# B&R Automation Studio project ProyectoDardos
Automation Studio 4.9

## Configuration Config1

CPU 4PPC70.0702-23B, AutomationRuntime B4.92, Build 4.1.2, Vc V4.72.5

### Task classes (Cpu.sw)
```
Cyclic#4:
  VisuCtrl <- Visu.VisuCtrl.prg
  ScoreCtrl <- Source.ScoreCtrl.prg
Cyclic#5 (cycle 250000 us, tolerance 250000 us):
  VisapiCtrl <- Source.VisapiCtrl.prg
VcDataObjects: VisuDa <- Visu.VisuDardos.dob
Binaries: vcnet, vccdbox, udbdef, vcrt, vcpkat, vcctext, vccurl, vcchtml, vccslider, visvc, vcfile, vcgclass, vccstr, vcpdsw, vccshape, arial, vccbmp, vcmgr, vcdsloc, VisuDa01, vcfntttf, vccovl, vcshared, arialbd, VisuDa02, VisuDa03, vcalarm, vccdt, vccline, vcpfar00, vccbtn, vcpdvnc, vcbclass, vcxml, vcdsint, vctcal, TCData, FWRules, vccnum, sysconf, iomap, asfw, Role, ashwac, ashwd, User, arconfig
Libraries: visapi, standard, vcresman, asieccon, fileio, astime, runtime, dataobj
```

### Hardware
```
4PPC70_0702_23B : 4PPC70.0702-23B v1.5.4.0
  Connector IF2:
    ActivateDevice = 1
    Mode = Manual
    InternetAddress = 192.168.150.95
    SubnetMask = 255.255.255.0
    Vnc1
    VncVcObjectName1 = VisuDa
    VncKeyMappingFile1 = VC\PS2-Keyboard.dis
    ActivateSnmp = 2
  ConfigurationID = proyectoDardos_Config1
  Cyclic5Duration = 250000
  Cyclic5Tolerance = 250000
  FileDevice1
  FileDeviceName1 = USER
  FileDevicePath1 = USER_PATH
  VcObjectName = VisuDa
  KeyMappingFile = VC\4PPC70_0702_23B.dis
```

## Logical view

### Global.typ - Global data types
```iecst
(*gMainCtrl_type*)

TYPE
	gMainCtrl_type : 	STRUCT
		visapiCtrl : visapiCtrl_type;
		scoreCtrl : scoreCtrl_type;
	END_STRUCT;
END_TYPE

(*visapiCtrl_type*)

TYPE
	visapiCtrl_type : 	STRUCT
		cmd : visapiCtrl_cmd_type;
		status : visapiCtrl_status_type;
		state : visapiCtrl_state_type;
	END_STRUCT;
	visapiCtrl_cmd_type : 	STRUCT
		readyToDraw : BOOL;
	END_STRUCT;
	visapiCtrl_status_type : 	STRUCT
		touchCoordinateX : REAL;
		drawing : BOOL;
		touchCoordinateY : REAL;
		valitTouch : BOOL;
		homeYCoordenate : REAL;
		homeXCoordenate : REAL;
		widthEllipse : ARRAY[1..6]OF UINT;
		heigthEllipse : ARRAY[1..6]OF UINT;
		widthTarget : UDINT;
		heigthTarget : UDINT;
		touchCoordinateStatus : BOOL;
		widthRect : UDINT;
	END_STRUCT;
	visapiCtrl_state_type :
		(
		WAIT := 0,
		DRAWING := 10,
		ERROR := 100
		);
END_TYPE

(*scoreCtrl_type*)

TYPE
	scoreCtrl_type : 	STRUCT
		cmd : scoreCtrl_cmd_type;
		status : scoreCtrl_status_type;
		state : scoreCtrl_state_type;
	END_STRUCT;
	scoreCtrl_cmd_type : 	STRUCT
		addPointScore : BOOL;
	END_STRUCT;
	scoreCtrl_status_type : 	STRUCT
		validTouch : BOOL;
		additivePoint : ARRAY[1..MAX_RADIUS_WITH_TARGET]OF UINT;
		incorrectScore : BOOL;
		correctScore : BOOL;
		cumulateScore : UINT;
		cumulateShots : UINT;
	END_STRUCT;
	scoreCtrl_state_type :
		(
		WAIT_SCORE := 0,
		GET_SCORE := 10,
		ERROR_SCORE := 100
		);
END_TYPE

(*gMachinePar*)

TYPE
	gMachinePar_type : 	STRUCT
		New_Member : USINT;
	END_STRUCT;
END_TYPE

(*gVisuCtrl_type*)

TYPE
	gVisuCtrl_type : 	STRUCT
		numInput : gVIsu_numInput_type;
		runtime : gVisu_runtime_type;
		button : gVisu_button_type;
		textOutput : gVisu_textOutput_type;
	END_STRUCT;
	gVIsu_numInput_type : 	STRUCT
		radiusWidth : ARRAY[1..MAX_RADIUS_WITH_TARGET]OF UINT;
		selectedRadiusWidth : ARRAY[1..MAX_RADIUS_WITH_TARGET]OF UINT;
	END_STRUCT;
	gVisu_runtime_type : 	STRUCT
		showButtonStartNewGame : USINT;
	END_STRUCT;
	gVisu_button_type : 	STRUCT
		startNewGame : BOOL;
	END_STRUCT;
	gVisu_textOutput_type : 	STRUCT
		statusGame : USINT;
	END_STRUCT;
END_TYPE
```

### Global.var - Global variables
```iecst
VAR
	gMainCtrl : gMainCtrl_type;
END_VAR
VAR RETAIN
	gMachinePar : {REDUND_UNREPLICABLE} gMachinePar_type := (0);
END_VAR
VAR CONSTANT
	LEFT_OFFSET : UINT := 28;
	TOP_OFFSET : UINT := 60;
	MAX_X_COORDINATE : UDINT := 434;
	MAX_Y_COORDINATE : UDINT := 413;
	MIN_X_COORDINATE : UDINT := 28;
	MIN_Y_COORDINATE : UDINT := 60;
	MAX_RADIUS : INT := 6;
	MAX_RADIUS_WITH_TARGET : UINT := 7;
END_VAR
VAR
	gVisuCtrl : gVisuCtrl_type;
END_VAR
VAR CONSTANT
	COORDENATE_Y_BITMAP : INT := 62;
	COORDENATE_X_BITMAP : INT := 358;
	MAX_SCORE : INT := 500;
	MAX_SHOTS : INT := 10;
END_VAR
```

### Program Logical/Source/ScoreCtrl (IEC)

#### Variables.var
```iecst
VAR
	getTouch : BOOL;
	homeXCoordenate : REAL;
	pointValue : UINT;
	ratio : REAL;
	homeYCoordenate : REAL;
	firstProduct : REAL;
	secondProduct : REAL;
END_VAR
VAR CONSTANT
	EXPONENT : INT := 2;
END_VAR
VAR
	intRatio : INT;
	countPointValue : UINT;
	valitPoint : BOOL;
	newTouch : BOOL;
	addPointsReady : BOOL;
	remainingShots : USINT;
END_VAR
VAR RETAIN
	maxShots : USINT;
	maxCountPointValue : INT;
END_VAR
VAR
	validCoordenate : BOOL;
	restorePointValues : BOOL;
	confirmValueRadius : BOOL;
END_VAR
(*AJUSTE DE PUNTAJES*)
VAR
	i : INT;
	actualRadius : INT;
	nextRadius : BOOL;
	previusRadius : BOOL;
	addivePoint : UINT;
END_VAR
```

#### Main.st
```iecst
PROGRAM _INIT
	actualRadius := 1;
	gMainCtrl.scoreCtrl.status.additivePoint[1] := 100;
	gMainCtrl.scoreCtrl.status.additivePoint[2] := 80;
	gMainCtrl.scoreCtrl.status.additivePoint[3] := 60;
	gMainCtrl.scoreCtrl.status.additivePoint[4] := 40;
	gMainCtrl.scoreCtrl.status.additivePoint[5] := 20;
	gMainCtrl.scoreCtrl.status.additivePoint[6] := 10;
	gMainCtrl.scoreCtrl.status.additivePoint[7] := 5;

END_PROGRAM

PROGRAM _CYCLIC
	homeXCoordenate := (gMainCtrl.visapiCtrl.status.homeXCoordenate);
	homeYCoordenate	:= (gMainCtrl.visapiCtrl.status.homeYCoordenate);
	newTouch		:= 	gMainCtrl.visapiCtrl.status.touchCoordinateStatus;

	firstProduct 	:= ABS(homeXCoordenate - gMainCtrl.visapiCtrl.status.touchCoordinateX);
	secondProduct	:= ABS(homeYCoordenate - gMainCtrl.visapiCtrl.status.touchCoordinateY);
	ratio := SQRT(EXPT(firstProduct,EXPONENT)+(EXPT(secondProduct,EXPONENT)));
	intRatio := REAL_TO_INT(ratio);

	IF restorePointValues THEN
		gMainCtrl.scoreCtrl.status.additivePoint[1] := 10;
		gMainCtrl.scoreCtrl.status.additivePoint[2] := 20;
		gMainCtrl.scoreCtrl.status.additivePoint[3] := 30;
		gMainCtrl.scoreCtrl.status.additivePoint[4] := 10;
		gMainCtrl.scoreCtrl.status.additivePoint[5] := 10;
		gMainCtrl.scoreCtrl.status.additivePoint[6] := 10;
		gMainCtrl.scoreCtrl.status.additivePoint[7] := 10;
	END_IF;

	///// AJUSTES DE PUNTAJE PARA CADA CIRCUNFERENCIA
	IF (actualRadius >= 1) AND (actualRadius <7) THEN
		IF EDGEPOS(nextRadius) THEN
			actualRadius:= actualRadius + 1;
		END_IF;
	END_IF;
	IF (actualRadius > 1) AND (actualRadius <= 7) THEN
		IF EDGEPOS(previusRadius) THEN
			actualRadius:= actualRadius - 1;
		END_IF;
	END_IF;

	IF actualRadius = 1 AND confirmValueRadius THEN
		confirmValueRadius := FALSE;
		gMainCtrl.scoreCtrl.status.additivePoint[1] := addivePoint;
	ELSIF actualRadius = 2 AND confirmValueRadius THEN
		confirmValueRadius := FALSE;
		gMainCtrl.scoreCtrl.status.additivePoint[2] := addivePoint;
	ELSIF actualRadius = 3 AND confirmValueRadius THEN
		confirmValueRadius := FALSE;
		gMainCtrl.scoreCtrl.status.additivePoint[3] := addivePoint;
	ELSIF actualRadius = 4 AND confirmValueRadius THEN
		confirmValueRadius := FALSE;
		gMainCtrl.scoreCtrl.status.additivePoint[4] := addivePoint;
	ELSIF actualRadius = 5 AND confirmValueRadius THEN
		confirmValueRadius := FALSE;
		gMainCtrl.scoreCtrl.status.additivePoint[5] := addivePoint;
	ELSIF actualRadius = 6 AND confirmValueRadius THEN
		confirmValueRadius := FALSE;
		gMainCtrl.scoreCtrl.status.additivePoint[6] := addivePoint;
	ELSIF actualRadius = 7 AND confirmValueRadius THEN
		confirmValueRadius := FALSE;
		gMainCtrl.scoreCtrl.status.additivePoint[7] := addivePoint;
	END_IF;

	IF	gMainCtrl.visapiCtrl.status.valitTouch THEN
		validCoordenate := TRUE;
	ELSE
		validCoordenate := FALSE;
	END_IF;

	CASE gMainCtrl.scoreCtrl.state OF

		WAIT_SCORE:

			IF EDGEPOS(newTouch) THEN
				IF (intRatio < gMainCtrl.visapiCtrl.status.widthRect) THEN
					gMainCtrl.scoreCtrl.cmd.addPointScore := TRUE;
					gMainCtrl.scoreCtrl.state	 := GET_SCORE;
				END_IF;
			END_IF;

		GET_SCORE:

			IF gMainCtrl.scoreCtrl.status.cumulateShots <= (MAX_SHOTS-1) AND gMainCtrl.scoreCtrl.cmd.addPointScore AND (gMainCtrl.scoreCtrl.status.cumulateScore < MAX_SCORE) AND validCoordenate THEN
				IF (intRatio <= gMainCtrl.visapiCtrl.status.heigthEllipse[1]/2) AND (intRatio > gMainCtrl.visapiCtrl.status.heigthEllipse[2]/2)  THEN
					gMainCtrl.scoreCtrl.cmd.addPointScore := FALSE;
					gMainCtrl.scoreCtrl.status.cumulateScore := gMainCtrl.scoreCtrl.status.cumulateScore  + gMainCtrl.scoreCtrl.status.additivePoint[7];
				ELSIF (intRatio <= gMainCtrl.visapiCtrl.status.heigthEllipse[2]/2) AND (intRatio > gMainCtrl.visapiCtrl.status.heigthEllipse[3]/2)  THEN
					gMainCtrl.scoreCtrl.cmd.addPointScore := FALSE;
					gMainCtrl.scoreCtrl.status.cumulateScore := gMainCtrl.scoreCtrl.status.cumulateScore + gMainCtrl.scoreCtrl.status.additivePoint[6];
				ELSIF (intRatio <= gMainCtrl.visapiCtrl.status.heigthEllipse[3]/2) AND (intRatio > gMainCtrl.visapiCtrl.status.heigthEllipse[4]/2)  THEN
					gMainCtrl.scoreCtrl.cmd.addPointScore := FALSE;
					pointValue := gMainCtrl.scoreCtrl.status.additivePoint[5];
					gMainCtrl.scoreCtrl.status.cumulateScore := gMainCtrl.scoreCtrl.status.cumulateScore + pointValue;
				ELSIF (intRatio <= gMainCtrl.visapiCtrl.status.heigthEllipse[4]/2) AND (intRatio > gMainCtrl.visapiCtrl.status.heigthEllipse[5]/2)  THEN
					gMainCtrl.scoreCtrl.cmd.addPointScore := FALSE;
					pointValue := gMainCtrl.scoreCtrl.status.additivePoint[4];
					gMainCtrl.scoreCtrl.status.cumulateScore := gMainCtrl.scoreCtrl.status.cumulateScore + pointValue;
				ELSIF (intRatio <= gMainCtrl.visapiCtrl.status.heigthEllipse[5]/2) AND (intRatio > gMainCtrl.visapiCtrl.status.heigthEllipse[6]/2)  THEN
					gMainCtrl.scoreCtrl.cmd.addPointScore := FALSE;
					pointValue := gMainCtrl.scoreCtrl.status.additivePoint[3];
					gMainCtrl.scoreCtrl.status.cumulateScore := gMainCtrl.scoreCtrl.status.cumulateScore + pointValue;
				ELSIF (intRatio <= gMainCtrl.visapiCtrl.status.heigthEllipse[6]/2) AND (intRatio > gMainCtrl.visapiCtrl.status.heigthTarget/2)  THEN
					gMainCtrl.scoreCtrl.cmd.addPointScore := FALSE;
					pointValue := gMainCtrl.scoreCtrl.status.additivePoint[2];
					gMainCtrl.scoreCtrl.status.cumulateScore := gMainCtrl.scoreCtrl.status.cumulateScore + pointValue;
				ELSIF (intRatio <= gMainCtrl.visapiCtrl.status.heigthTarget/2)  THEN
					gMainCtrl.scoreCtrl.cmd.addPointScore := FALSE;
					pointValue := gMainCtrl.scoreCtrl.status.additivePoint[1];
					gMainCtrl.scoreCtrl.status.cumulateScore := gMainCtrl.scoreCtrl.status.cumulateScore + pointValue;
				ELSIF (intRatio > gMainCtrl.visapiCtrl.status.heigthEllipse[1]/2) AND (gMainCtrl.scoreCtrl.cmd.addPointScore )(* AND (gMainCtrl.scoreCtrl.status.cumulateShots <= (MAX_SHOTS-1))*) THEN
					gMainCtrl.scoreCtrl.cmd.addPointScore := FALSE;
				END_IF;

				gMainCtrl.scoreCtrl.status.cumulateShots := gMainCtrl.scoreCtrl.status.cumulateShots + 1;

			END_IF;

			IF 	intRatio > (gMainCtrl.visapiCtrl.status.heigthEllipse[1]/2) THEN
				gMainCtrl.scoreCtrl.status.incorrectScore := TRUE;
				gMainCtrl.scoreCtrl.status.correctScore := FALSE;
			ELSIF (intRatio <= gMainCtrl.visapiCtrl.status.heigthEllipse[1]/2) THEN
				gMainCtrl.scoreCtrl.status.correctScore := TRUE;
				gMainCtrl.scoreCtrl.status.incorrectScore := FALSE;
			END_IF

			IF EDGENEG(newTouch) THEN
				gMainCtrl.scoreCtrl.state	 := WAIT_SCORE;
			END_IF;

	END_CASE;

END_PROGRAM

PROGRAM _EXIT
			(* Insert code here *)

END_PROGRAM
```

### Program Logical/Source/VisapiCtrl (IEC)

#### Types.typ
```iecst
TYPE
	VA_SetupX_0 : 	STRUCT
		enable : BOOL;
		VCHandle : VCHANDLE;
		interpreter : STRING[80] := 'VisuDa';
		status : UINT;
	END_STRUCT;
	VA_Saccess_0 : 	STRUCT
		enable : BOOL;
		VCHandle : VCHANDLE;
		status : UINT;
	END_STRUCT;
END_TYPE
```

#### Variables.var
```iecst
(*VISAPI*)
VAR
	ready : UINT;
	VC_HANDLE : UDINT;
	interpreter : STRING[80] := 'VisuDa';
END_VAR
(*VA_Rect*)
VAR
	xRect : ARRAY[1..MAX_RECT] OF UINT := [28,0,229]; (*coordenada X del rectangulo*)
	yRect : ARRAY[1..MAX_RECT] OF UINT := [60,235,0]; (*coordenada Y del rectangulo*)
	widthRect : ARRAY[1..MAX_RECT] OF UINT := [406,0,4]; (*ancho del rectangulo*)
	heigthRect : ARRAY[1..MAX_RECT] OF UINT := [353,4,0]; (*altura del rectangulo*)
	fillRect : ARRAY[1..MAX_RECT] OF UINT := [255,2(45)]; (*relleno del rectangulo*)
	colorRect : ARRAY[1..MAX_RECT] OF UINT := [255,2(45)]; (*contorno del rectanculo*)
END_VAR
(*VA_Ellipse*)
VAR CONSTANT
	xEllipse : UINT := 231; (*coordenada X de la elipse*)
	yEllipse : UINT := 237; (*coordenadas Y de la elipse*)
END_VAR
VAR RETAIN
	heigthEllipse : ARRAY[1..MAX_RADIUS] OF UINT; (*altura de la elipse*)
	widthEllipse : ARRAY[1..MAX_RADIUS] OF UINT; (*ancho de la elipse*)
END_VAR
VAR
	fillEllipse : ARRAY[1..MAX_RADIUS] OF UINT := [45,16,45,16,45,16]; (*relleno de la elipse*)
END_VAR
VAR RETAIN
	colorEllipse : ARRAY[1..MAX_RADIUS] OF UINT := [0,16,45,16,45,16]; (*contorno de la elipse*)
END_VAR
VAR CONSTANT
	xTarget : UINT := 231; (*coordenada X del target*)
	yTarget : UINT := 237; (*coordenada Y del target*)
END_VAR
VAR
	heigthTarget : UINT;
	widthTarget : UINT;
	fillTarget : USINT := 205;
	colorTarget : USINT := 45;
	updateRadio : UINT;
END_VAR
(*AUX *)
VAR
	actualPage : UINT; (*pagina actual*)
	j : INT;
	defaultRadiusValues : BOOL;
END_VAR
VAR CONSTANT
	MAX_RECT : INT := 3;
END_VAR
(*VA_GetTouchAction*)
VAR
	xTouchPosition : UDINT;
	yTouchPosition : UDINT;
	Touch : TouchAction;
	newTouch : BOOL;
	changeRatioValue : BOOL;
	actualRadius : INT;
	nextRadius : BOOL;
	previusRadius : BOOL;
	confirmValueRadius : BOOL;
END_VAR
```

#### Main.st
```iecst
PROGRAM _INIT
	//Inicialización de circunferencias
	gMainCtrl.visapiCtrl.status.heigthEllipse[1] := 330;
	gMainCtrl.visapiCtrl.status.heigthEllipse[2] := 280;
	gMainCtrl.visapiCtrl.status.heigthEllipse[3] := 230;
	gMainCtrl.visapiCtrl.status.heigthEllipse[4] := 180;
	gMainCtrl.visapiCtrl.status.heigthEllipse[5] := 130;
	gMainCtrl.visapiCtrl.status.heigthEllipse[6] := 80;
	gMainCtrl.visapiCtrl.status.heigthTarget	 := 40;
	heigthTarget	 := 30;
	xTouchPosition;
	yTouchPosition;
	actualRadius := 1;
END_PROGRAM

PROGRAM _CYCLIC

	FOR j:= 1 TO MAX_RADIUS DO
		heigthEllipse[j] := gMainCtrl.visapiCtrl.status.heigthEllipse[j];
		widthEllipse[j] := gMainCtrl.visapiCtrl.status.widthEllipse[j];
	END_FOR;

	//CORDENADAS, ALTO Y ANCHO DE LOS RECTANGULOS QUE DIVIDEN EL TABLERO
	xRect[2]:= ((widthRect[1]/2)-(gMainCtrl.visapiCtrl.status.widthEllipse[1]/2))+ LEFT_OFFSET;
	yRect[3]:=((heigthRect[1]/2)-(gMainCtrl.visapiCtrl.status.widthEllipse[1]/2))+ TOP_OFFSET;
	widthRect[2] := gMainCtrl.visapiCtrl.status.widthEllipse[1];
	heigthRect[3] := gMainCtrl.visapiCtrl.status.widthEllipse[1];
	widthTarget	:= heigthTarget;

	IF defaultRadiusValues THEN
		gMainCtrl.visapiCtrl.status.heigthEllipse[1] := 330;
		gMainCtrl.visapiCtrl.status.heigthEllipse[2] := 280;
		gMainCtrl.visapiCtrl.status.heigthEllipse[3] := 230;
		gMainCtrl.visapiCtrl.status.heigthEllipse[4] := 180;
		gMainCtrl.visapiCtrl.status.heigthEllipse[5] := 130;
		gMainCtrl.visapiCtrl.status.heigthEllipse[6] := 80;
		gMainCtrl.visapiCtrl.status.heigthTarget	 := 40;
	END_IF;

	IF Touch.status = 1 THEN
		newTouch 	:= TRUE;
	ELSE
		newTouch	:= FALSE;
	END_IF;

	///// AJUSTES DE PUNTAJE PARA CADA CIRCUNFERENCIA
	IF (actualRadius >= 1) AND (actualRadius <7) THEN
		IF EDGEPOS(nextRadius) THEN
			actualRadius:= actualRadius + 1;
		END_IF;
	END_IF;
	IF (actualRadius > 1) AND (actualRadius <= 7) THEN
		IF EDGEPOS(previusRadius) THEN
			actualRadius:= actualRadius - 1;
		END_IF;
	END_IF;

	IF actualRadius = 1 AND confirmValueRadius THEN
		confirmValueRadius := FALSE;
		heigthTarget		:= updateRadio;
	ELSIF actualRadius = 2 AND confirmValueRadius THEN
		confirmValueRadius := FALSE;
		gMainCtrl.visapiCtrl.status.heigthEllipse[6] := updateRadio;
	ELSIF actualRadius = 3 AND confirmValueRadius THEN
		confirmValueRadius := FALSE;
		gMainCtrl.visapiCtrl.status.heigthEllipse[5] := updateRadio;
	ELSIF actualRadius = 4 AND confirmValueRadius THEN
		confirmValueRadius := FALSE;
		gMainCtrl.visapiCtrl.status.heigthEllipse[4] := updateRadio;
	ELSIF actualRadius = 5 AND confirmValueRadius THEN
		confirmValueRadius := FALSE;
		gMainCtrl.visapiCtrl.status.heigthEllipse[3] := updateRadio;
	ELSIF actualRadius = 6 AND confirmValueRadius THEN
		confirmValueRadius := FALSE;
		gMainCtrl.visapiCtrl.status.heigthEllipse[2] := updateRadio;
	ELSIF actualRadius = 7 AND confirmValueRadius THEN
		confirmValueRadius := FALSE;
		gMainCtrl.visapiCtrl.status.heigthEllipse[1] := updateRadio;
	END_IF;

	CASE gMainCtrl.visapiCtrl.state OF

		WAIT:
			IF ready <> 1 THEN
				VC_HANDLE := VA_Setup(1,interpreter);
				ready := 1;
			END_IF;
			IF  (*oldHeight <> height AND*) ready = 1 THEN
				gMainCtrl.visapiCtrl.state := DRAWING;
			END_IF;

		DRAWING:

			IF ready = 1 AND actualPage = 0 THEN
				IF VA_Saccess(1, VC_HANDLE) = 0 THEN

					IF changeRatioValue THEN
						changeRatioValue	:= FALSE;
						VA_Redraw(1,VC_HANDLE);
					END_IF;

					VA_Rect(1,VC_HANDLE,xRect[1],yRect[1],widthRect[1],heigthRect[1],fillRect[1],colorRect[1]);

					FOR j:= 1 TO (MAX_RADIUS) DO
						fillEllipse[j+1]	:= colorEllipse[j+1];
						gMainCtrl.visapiCtrl.status.widthEllipse[j] := gMainCtrl.visapiCtrl.status.heigthEllipse[j];
						VA_Ellipse(1,VC_HANDLE,xEllipse ,yEllipse,gMainCtrl.visapiCtrl.status.heigthEllipse[j] ,gMainCtrl.visapiCtrl.status.widthEllipse[j],fillEllipse[j],colorEllipse[j]);
					END_FOR;

					VA_Rect(1,VC_HANDLE,xRect[2],yRect[2],widthRect[2],heigthRect[2],fillRect[2],colorRect[2]); //RECTANGULO HORIZONTAL
					VA_Rect(1,VC_HANDLE,xRect[3],yRect[3],widthRect[3],heigthRect[3],fillRect[3],colorRect[3]); //RECTANGULO VERTICAL
					VA_Ellipse(1,VC_HANDLE,xTarget,yTarget,heigthTarget,widthTarget,fillTarget,colorTarget); //TARGET
					VA_GetTouchAction(1,VC_HANDLE,0,ADR(Touch)); //COORDENADAS DEL TOUCH

					IF gMainCtrl.scoreCtrl.status.cumulateShots < MAX_SHOTS THEN
						IF EDGEPOS(gMainCtrl.scoreCtrl.status.incorrectScore) AND (gMainCtrl.visapiCtrl.status.valitTouch) THEN
							gMainCtrl.visapiCtrl.status.valitTouch := FALSE;
							VA_DrawBitmap(1,VC_HANDLE,1421,COORDENATE_X_BITMAP,COORDENATE_Y_BITMAP);

						ELSIF EDGEPOS(gMainCtrl.scoreCtrl.status.correctScore) AND (gMainCtrl.visapiCtrl.status.valitTouch) THEN
							gMainCtrl.visapiCtrl.status.valitTouch := FALSE;
							VA_DrawBitmap(1,VC_HANDLE,1420,COORDENATE_X_BITMAP,COORDENATE_Y_BITMAP);
						END_IF;
					END_IF

					VA_Srelease(1, VC_HANDLE);
				END_IF;
			END_IF;

			//RESET VA_SETUP EN CASO DE ERROR
			IF VC_HANDLE = 0 THEN
				gMainCtrl.visapiCtrl.state := ERROR;
			END_IF;

		ERROR:
			gMainCtrl.visapiCtrl.state := WAIT;

	END_CASE;

	//SENTENCIA PARA CONSIDERAR UN TOQUE EN EL AREA DE JUEGO
	IF Touch.x <= MAX_X_COORDINATE AND (Touch.x >= MIN_X_COORDINATE) AND(Touch.y <= MAX_Y_COORDINATE) AND(Touch.y >= MIN_Y_COORDINATE)
		AND (Touch.status = 1) THEN
		gMainCtrl.visapiCtrl.status.valitTouch := TRUE;
	ELSE
		gMainCtrl.visapiCtrl.status.valitTouch := FALSE;
	END_IF;

	//CONEXION DE VARIABLES LOCALES A GLOBALES
	gMainCtrl.visapiCtrl.status.widthRect				:= widthRect[1];
	gMainCtrl.visapiCtrl.status.widthTarget 			:= widthTarget;
	gMainCtrl.visapiCtrl.status.heigthTarget			:= heigthTarget;
	gMainCtrl.visapiCtrl.status.homeXCoordenate 		:= UDINT_TO_REAL (xTarget);
	gMainCtrl.visapiCtrl.status.homeYCoordenate			:= UDINT_TO_REAL (yTarget);
	gMainCtrl.visapiCtrl.status.touchCoordinateX 		:= UDINT_TO_REAL (Touch.x);
	gMainCtrl.visapiCtrl.status.touchCoordinateY 		:= UDINT_TO_REAL (Touch.y);
	gMainCtrl.visapiCtrl.status.touchCoordinateStatus	:= newTouch;
END_PROGRAM

PROGRAM _EXIT
	(* Insert code here *)

END_PROGRAM
```

- Visualisation Logical/Visu (not shown)

Listed in the project but not available here: Logical/Libraries
